FUNCTION Convert_ULINT_TO_BOOL : Hresult
VAR_INPUT
	in : ULINT;
	out : REFERENCE TO BOOL;
END_VAR
VAR
	converted : BOOL;
END_VAR
VAR CONSTANT
	INCOMPATIBLE : HRESULT := 16#9811070E;
END_VAR

converted := ULINT_TO_BOOL(in);

IF (BOOL_TO_ULINT(converted) <> in) THEN
	Convert_ULINT_TO_BOOL := INCOMPATIBLE;
	RETURN;
END_IF

out := converted;

END_FUNCTION

(* stored: Version 1.1.0.1, ProductVersion 3.1.4024.12
   POU Convert_ULINT_TO_BOOL: Id {1def3589-cc70-4ab3-9ff5-18ff02b0870b}, SpecialFunc None *)
